{attribute 'qualified_only'}
VAR_GLOBAL
    stBasicMotor: DUT_MotionStage;
END_VAR

(* stored: Version 1.1.0.1, ProductVersion 3.1.4022.18
   GVL SIM: Id {c2b1c90b-ecac-4fe0-9807-d60159bc2e98} *)
